FUNCTION_BLOCK ProjectSpecificData EXTENDS TcoCognexVision.TcoDesignerRootContainer
VAR_INPUT
END_VAR
VAR_OUTPUT
END_VAR
VAR
    {attribute wpf [Container(Layout.Stack,"PcToPlc")]}
    {attribute wpf [Group(Layout.GroupBox)]}
    {attribute addProperty Name "<#PcToPlc#>"}
    PcToPlc : DesignerResults;
    {attribute wpf [Container(Layout.Stack,"PlcToPc")]}
    {attribute wpf [Group(Layout.GroupBox)]}
    {attribute addProperty Name "<#PlcToPc#>"}
    PlcToPc : DesignerUserData;
END_VAR

PROPERTY PUBLIC Results : REFERENCE TO DesignerResults
GET
Results ref= PcToPlc;
END_GET
END_PROPERTY

PROPERTY PUBLIC UserData : REFERENCE TO DesignerUserData
GET
UserData ref= PlcToPc;
END_GET
END_PROPERTY

END_FUNCTION_BLOCK

(* stored: Version 1.1.0.1, ProductVersion 3.1.4024.12
   POU ProjectSpecificData: Id {b6e257e8-4495-0a98-09f7-b4bfa71f5dc6}, SpecialFunc None
   Property Results: Id {c6f044b0-d898-0b05-2ec5-b2833a02c0f3}
   Get Get: Id {55dfda30-672c-0423-3bd8-a7a552c928c7}
   Property UserData: Id {fa3036d3-b0eb-02b7-37f7-b0bd32efe0ed}
   Get Get: Id {54b5f4cf-7a98-07f9-19d9-fdf4e0978468} *)
